// TIA Portal V20 export
FUNCTION_BLOCK "SysCounterFast"   // FB2035, FBD
TITLE = manage a incremental encoder conected to a counter module
{ S7_Optimized_Access := 'TRUE' }
AUTHOR : MiCROTEC
VERSION : 1.6
// -2018.09 : Martin
// -2019.10 : Martin
// stored: AutoNumber false, MemoryReserve 100, SetENOAutomatically false
   VAR_INPUT
      adr { ExternalAccessible := 'False'; ExternalVisible := 'False'; ExternalWritable := 'False'} : HW_IO;   // I/O adresse
      changeDir { ExternalAccessible := 'False'; ExternalVisible := 'False'; ExternalWritable := 'False'} : Bool;   // change direction
      reset { ExternalAccessible := 'False'; ExternalVisible := 'False'; ExternalWritable := 'False'} : Bool;   // reset counter
      calOffset { ExternalAccessible := 'False'; ExternalVisible := 'False'; ExternalWritable := 'False'} : Real;   // offset [mm], the "Reset" will take effect after the offset value
      calGain { ExternalAccessible := 'False'; ExternalVisible := 'False'; ExternalWritable := 'False'} : Real;   // gain
      set { ExternalAccessible := 'False'; ExternalVisible := 'False'; ExternalWritable := 'False'} : Bool;   // set counter on "set value"
      setValue { ExternalAccessible := 'False'; ExternalVisible := 'False'; ExternalWritable := 'False'} : Real;   // set value [mm]
      ack { ExternalAccessible := 'False'; ExternalVisible := 'False'; ExternalWritable := 'False'} : Bool;   // fault acknowledge
      runCheckActive { ExternalAccessible := 'False'; ExternalVisible := 'False'; ExternalWritable := 'False'} : Bool;   // activate plausibility check of encoder value and run signal
      runCheckTime { ExternalAccessible := 'False'; ExternalVisible := 'False'; ExternalWritable := 'False'} : Time := T#3S;   // run signal check fault time
      runCheckDiff { ExternalAccessible := 'False'; ExternalVisible := 'False'; ExternalWritable := 'False'} : Real := 0.5;   // difference value for run check
      runSig { ExternalAccessible := 'False'; ExternalVisible := 'False'; ExternalWritable := 'False'} : Bool;   // run signal for drive
      errOffDelTime { ExternalAccessible := 'False'; ExternalVisible := 'False'; ExternalWritable := 'False'} : Time := T#1S;   // err off delayed time
      limMin { ExternalAccessible := 'False'; ExternalVisible := 'False'; ExternalWritable := 'False'} : Real;   // minimum limit position (0 = deactivated )
      limMax { ExternalAccessible := 'False'; ExternalVisible := 'False'; ExternalWritable := 'False'} : Real;   // maximum limit position (0 = deactivated )
   END_VAR
   VAR_OUTPUT
      comOk { ExternalAccessible := 'False'; ExternalVisible := 'False'; ExternalWritable := 'False'} : Bool;   // communication ok/active
      ready { ExternalAccessible := 'False'; ExternalVisible := 'False'; ExternalWritable := 'False'} : Bool;   // ready to work
      encAct { ExternalAccessible := 'False'; ExternalVisible := 'False'; ExternalWritable := 'False'} : DInt;   // actual position from counter
      delta { ExternalAccessible := 'False'; ExternalVisible := 'False'; ExternalWritable := 'False'} : Real;   // delta in millimeter
      resetPos { ExternalAccessible := 'False'; ExternalVisible := 'False'; ExternalWritable := 'False'} : Real;   // last reset position for the encoder value (ex. division sensor)
      act { ExternalAccessible := 'False'; ExternalVisible := 'False'; ExternalWritable := 'False'} : Real;   // actual position in millimeter
      sync { ExternalAccessible := 'False'; ExternalVisible := 'False'; ExternalWritable := 'False'} : Bool;   // reset puls (division sensor, or generate with offset)
      err { ExternalAccessible := 'False'; ExternalVisible := 'False'; ExternalWritable := 'False'} : Bool;   // fault
      errCom { ExternalAccessible := 'False'; ExternalVisible := 'False'; ExternalWritable := 'False'} : Bool;   // fault communication
      errRdEnc { ExternalAccessible := 'False'; ExternalVisible := 'False'; ExternalWritable := 'False'} : Bool;   // fault encoder from count module
      errRunCheck { ExternalAccessible := 'False'; ExternalVisible := 'False'; ExternalWritable := 'False'} : Bool;   // fault plausibility check run-signal/encoder-value
      errLim { ExternalAccessible := 'False'; ExternalVisible := 'False'; ExternalWritable := 'False'} : Bool;   // fault position is outside from limits
      errOverFlow { ExternalAccessible := 'False'; ExternalVisible := 'False'; ExternalWritable := 'False'} : Bool;   // fault implausible change in encoder value detected (maybe overflow or underflow)
   END_VAR
   VAR_IN_OUT
      Enc : "TypeEncoder";
   END_VAR
   VAR
      var { ExternalAccessible := 'False'; ExternalVisible := 'False'; ExternalWritable := 'False'; S7_SetPoint := 'True'} : "TypeVar";
      T { ExternalAccessible := 'False'; ExternalVisible := 'False'; ExternalWritable := 'False'; S7_SetPoint := 'True'} : Array[1..3] of IEC_TIMER;
      Rd { ExternalAccessible := 'False'; ExternalVisible := 'False'; ExternalWritable := 'False'} : Struct
         cntBit24 : Bool;   // count value
         stsDI1 : Bool;   // DI1 status
         stsDir : Bool;   // direction
         stsDI0 : Bool;   // DI0 status
         err : Bool;   // fault
         stsDI2 : Bool;   // Tm Count: status DI2
         stsReady : Bool;   // ready
         Wd : Bool;   // watchdog if used isochronous mode
         cntValue2 : Byte;   // count value
         cntValue : Word;   // count value
      END_STRUCT;
      encActOld { ExternalAccessible := 'False'; ExternalVisible := 'False'; ExternalWritable := 'False'} : DInt;
      deltaIncOld { ExternalAccessible := 'False'; ExternalVisible := 'False'; ExternalWritable := 'False'} : DInt;
      actualNoOffset { ExternalAccessible := 'False'; ExternalVisible := 'False'; ExternalWritable := 'False'} : Real;
      errLimMin { ExternalAccessible := 'False'; ExternalVisible := 'False'; ExternalWritable := 'False'} : Bool;
      errLimMax { ExternalAccessible := 'False'; ExternalVisible := 'False'; ExternalWritable := 'False'} : Bool;
   END_VAR
   VAR_TEMP
      tempDelta1 : DInt;
      tempRdRetVal : Int;
      tempErrOverFlow : Bool;
   END_VAR
   VAR_TEMP   // added for the SCL form of the ladder/FBD networks
      _w1 : Bool;
      _w2 : Bool;
   END_VAR
BEGIN

REGION Network 1: exit
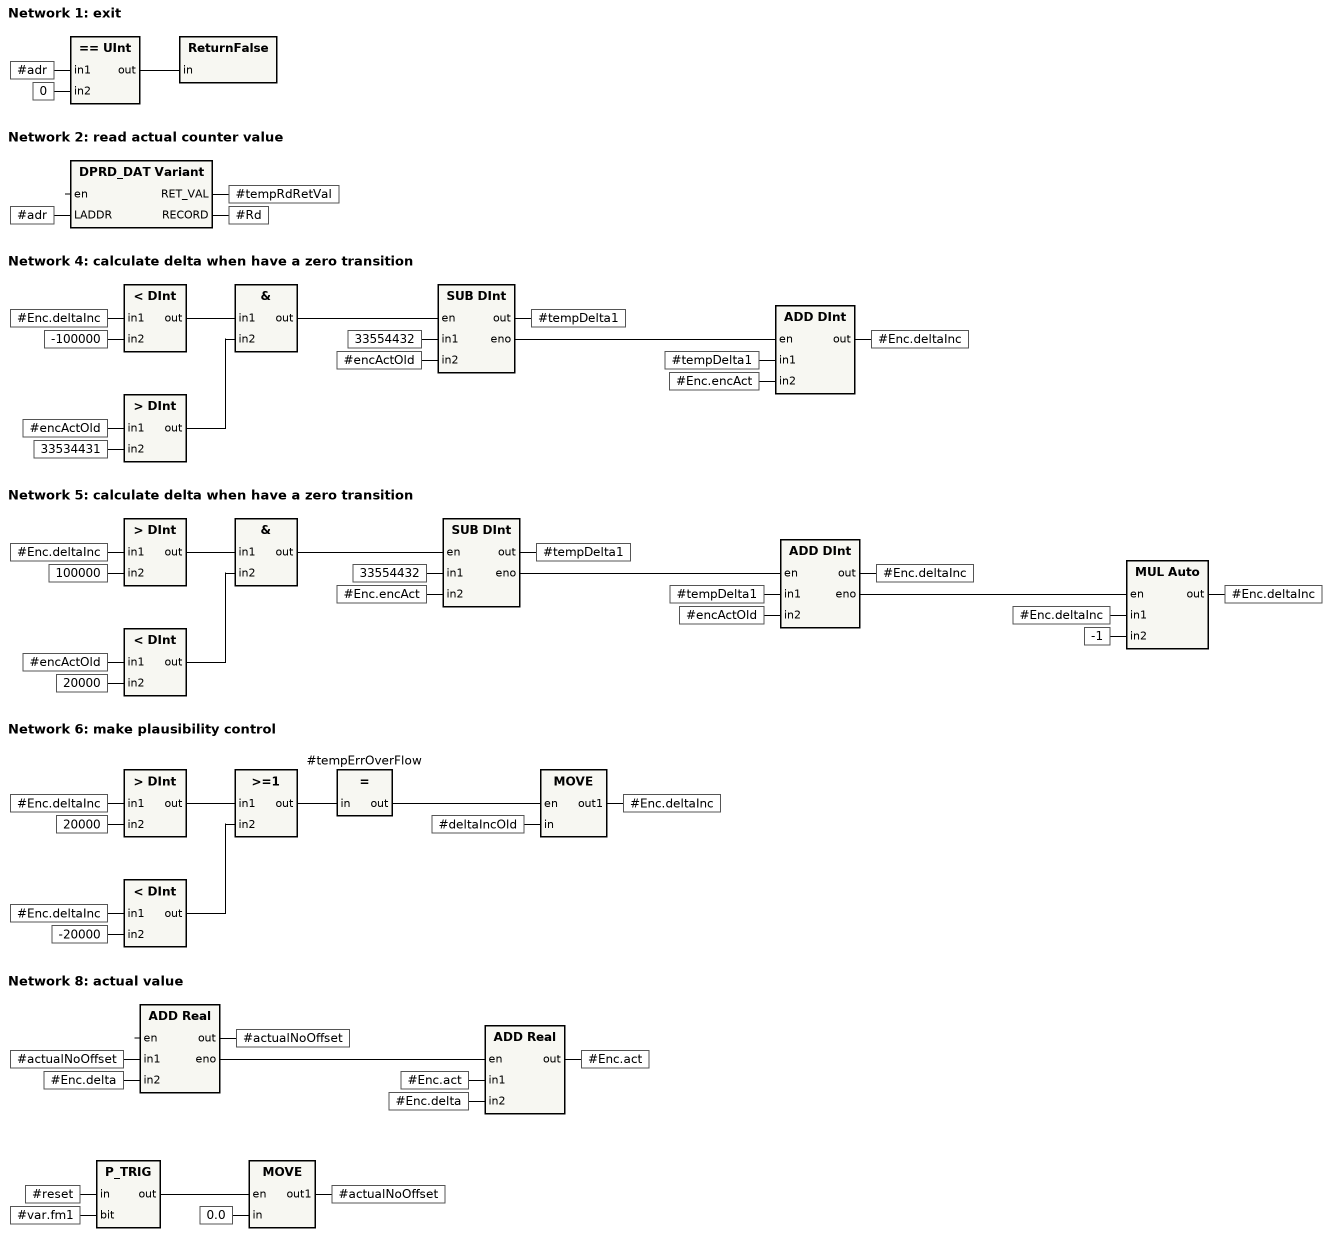
   IF #adr = 0 THEN
       ENO := FALSE;
       RETURN;
   END_IF;
END_REGION

REGION Network 2: read actual counter value
   #tempRdRetVal := DPRD_DAT(LADDR := #adr, RECORD => #Rd);
END_REGION

REGION Network 3 (SCL): read/write values

   #Enc.ready := #Rd.stsReady;
   #Enc.encAct :=  WORD_TO_DWORD(#Rd.cntValue) OR SHL_DWORD(IN:=BYTE_TO_DWORD(#Rd.cntValue2), N:=16);
   #Enc.encAct.%X24 := #Rd.cntBit24;
   #Enc.calOffset := #calOffset;
   #Enc.refPos := #setValue;
   #Enc.limMin := #limMin;
   #Enc.limMax := #limMax;
   #Enc.dirUp := #Rd.stsDir;
   #Enc.dirDn := NOT #Rd.stsDir;

   IF #calGain <> 0.0 THEN
       #Enc.calGain := #calGain;
   ELSE
       #Enc.calGain := 1.0;
   END_IF;

   #Enc.deltaInc := #Enc.encAct - #encActOld;
END_REGION

REGION Network 4: calculate delta when have a zero transition
   // ENO of a box is taken as its EN; it also drops when the box reports an error
   IF (#Enc.deltaInc < (-100000)) AND (#encActOld > 33534431) THEN
       #tempDelta1 := 33554432 - #encActOld;
       #Enc.deltaInc := #tempDelta1 + #Enc.encAct;
   END_IF;
END_REGION

REGION Network 5: calculate delta when have a zero transition
   // ENO of a box is taken as its EN; it also drops when the box reports an error
   IF (#Enc.deltaInc > 100000) AND (#encActOld < 20000) THEN #tempDelta1 := 33554432 - #Enc.encAct; END_IF;
   #_w1 := (#Enc.deltaInc > 100000) AND (#encActOld < 20000);
   IF #_w1 THEN
       #Enc.deltaInc := #tempDelta1 + #encActOld;
       #Enc.deltaInc := #Enc.deltaInc * (-1);
   END_IF;
END_REGION

REGION Network 6: make plausibility control
   #tempErrOverFlow := (#Enc.deltaInc > 20000) OR (#Enc.deltaInc < (-20000));
   IF #tempErrOverFlow THEN #Enc.deltaInc := #deltaIncOld; END_IF;
END_REGION

REGION Network 7 (SCL): increment in mm and actual speed in meter/min
   #Enc.delta := DINT_TO_REAL( #Enc.deltaInc) * #Enc.calGain;
   #Enc.speed := #Enc.speed * 0.9 + (#Enc.delta * 60.0 / "cycle") * 0.1;

   //save old value
   #deltaIncOld := #Enc.deltaInc;
   #encActOld := #Enc.encAct;
END_REGION

REGION Network 8: actual value
   // ENO of a box is taken as its EN; it also drops when the box reports an error
   #actualNoOffset := #actualNoOffset + #Enc.delta;
   #Enc.act := #Enc.act + #Enc.delta;
   #_w1 := #reset AND NOT #var.fm1;   // rising edge
   #var.fm1 := #reset;
   IF #_w1 THEN #actualNoOffset := 0.0; END_IF;
END_REGION

REGION Network 9: virtual reset
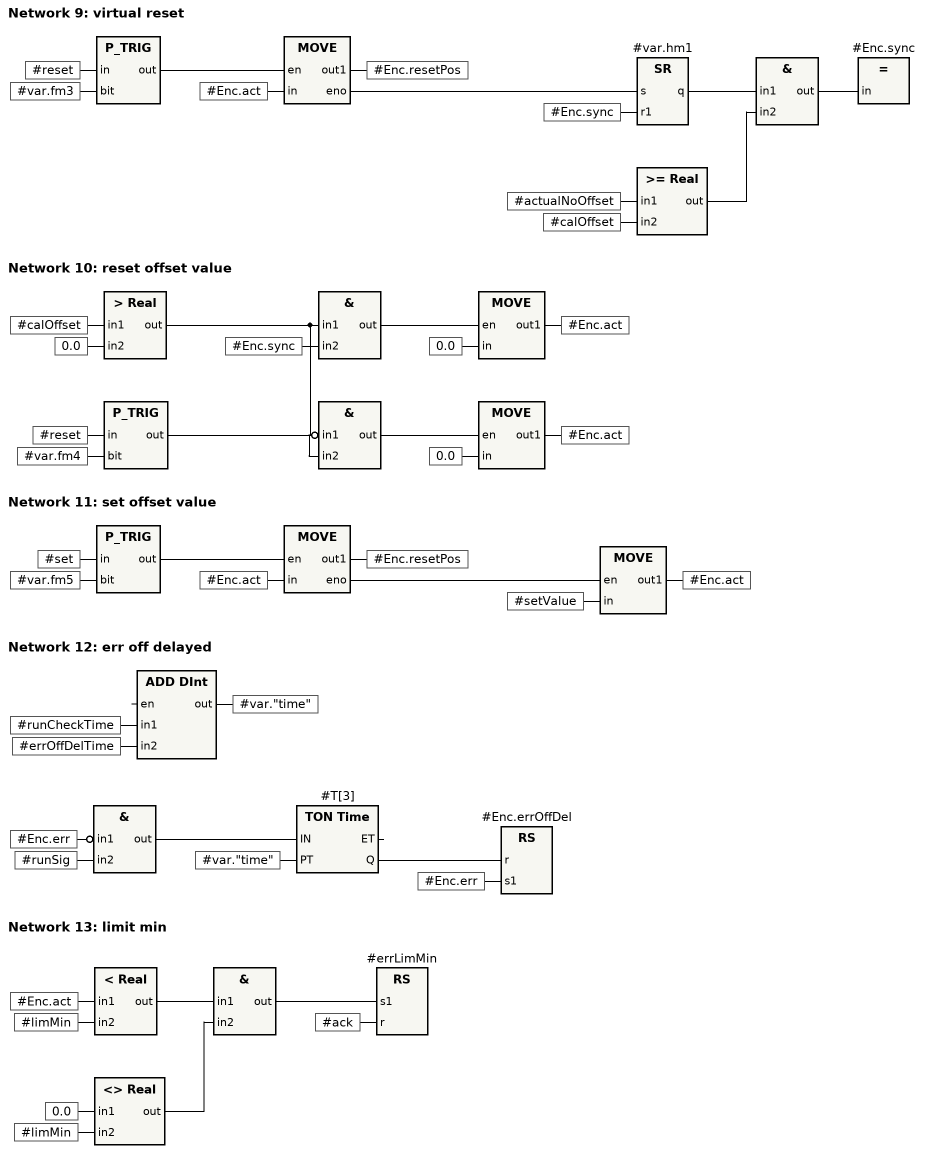
   #_w1 := #reset AND NOT #var.fm3;   // rising edge
   #var.fm3 := #reset;
   IF #_w1 THEN
       #Enc.resetPos := #Enc.act;
       #var.hm1 := TRUE;   // SR flip-flop
   END_IF;
   IF #Enc.sync THEN #var.hm1 := FALSE; END_IF;
   #Enc.sync := #var.hm1 AND (#actualNoOffset >= #calOffset);
END_REGION

REGION Network 10: reset offset value
   #_w1 := #calOffset > 0.0;
   IF #_w1 AND #Enc.sync THEN #Enc.act := 0.0; END_IF;
   #_w2 := #reset AND NOT #var.fm4;   // rising edge
   #var.fm4 := #reset;
   IF NOT #_w1 AND #_w2 THEN #Enc.act := 0.0; END_IF;
END_REGION

REGION Network 11: set offset value
   #_w1 := #set AND NOT #var.fm5;   // rising edge
   #var.fm5 := #set;
   IF #_w1 THEN
       #Enc.resetPos := #Enc.act;
       #Enc.act := #setValue;
   END_IF;
END_REGION

REGION Network 12: err off delayed
   #var."time" := #runCheckTime + #errOffDelTime;
   #T[3].TON(IN := NOT #Enc.err AND #runSig, PT := #var."time");
   IF #T[3].Q THEN
       #Enc.errOffDel := FALSE;   // RS flip-flop
   END_IF;
   IF #Enc.err THEN #Enc.errOffDel := TRUE; END_IF;
END_REGION

REGION Network 13: limit min
   IF #ack THEN
       #errLimMin := FALSE;   // RS flip-flop
   END_IF;
   IF (#Enc.act < #limMin) AND (0.0 <> #limMin) THEN #errLimMin := TRUE; END_IF;
END_REGION

REGION Network 14: limit max
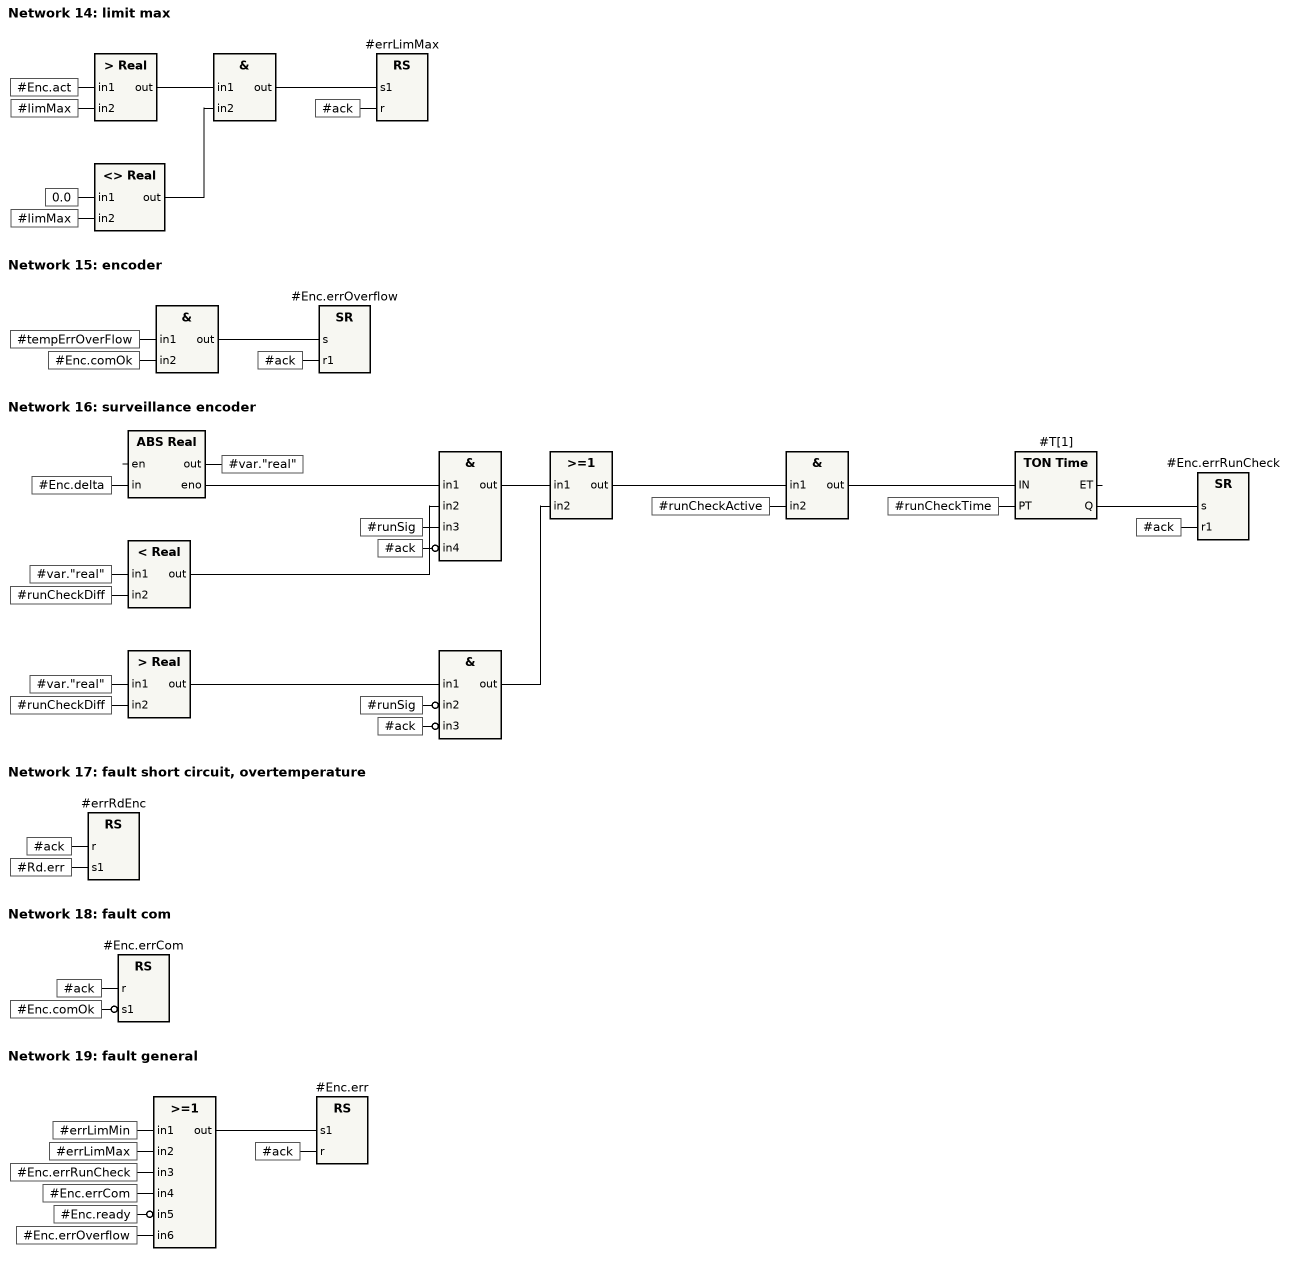
   IF #ack THEN
       #errLimMax := FALSE;   // RS flip-flop
   END_IF;
   IF (#Enc.act > #limMax) AND (0.0 <> #limMax) THEN #errLimMax := TRUE; END_IF;
END_REGION

REGION Network 15: encoder
   IF #tempErrOverFlow AND #Enc.comOk THEN
       #Enc.errOverflow := TRUE;   // SR flip-flop
   END_IF;
   IF #ack THEN #Enc.errOverflow := FALSE; END_IF;
END_REGION

REGION Network 16: surveillance encoder
   #var."real" := ABS(#Enc.delta);
   #T[1].TON(IN := (((#var."real" < #runCheckDiff) AND #runSig AND NOT #ack) OR ((#var."real" > #runCheckDiff) AND NOT #runSig AND NOT #ack)) AND #runCheckActive,
             PT := #runCheckTime);
   IF #T[1].Q THEN
       #Enc.errRunCheck := TRUE;   // SR flip-flop
   END_IF;
   IF #ack THEN #Enc.errRunCheck := FALSE; END_IF;
END_REGION

REGION Network 17: fault short circuit, overtemperature
   IF #ack THEN
       #errRdEnc := FALSE;   // RS flip-flop
   END_IF;
   IF #Rd.err THEN #errRdEnc := TRUE; END_IF;
END_REGION

REGION Network 18: fault com
   IF #ack THEN
       #Enc.errCom := FALSE;   // RS flip-flop
   END_IF;
   IF NOT #Enc.comOk THEN #Enc.errCom := TRUE; END_IF;
END_REGION

REGION Network 19: fault general
   IF #ack THEN
       #Enc.err := FALSE;   // RS flip-flop
   END_IF;
   IF #errLimMin OR #errLimMax OR #Enc.errRunCheck OR #Enc.errCom OR NOT #Enc.ready OR #Enc.errOverflow THEN
       #Enc.err := TRUE;
   END_IF;
END_REGION

REGION Network 20: error number counter [1-50]
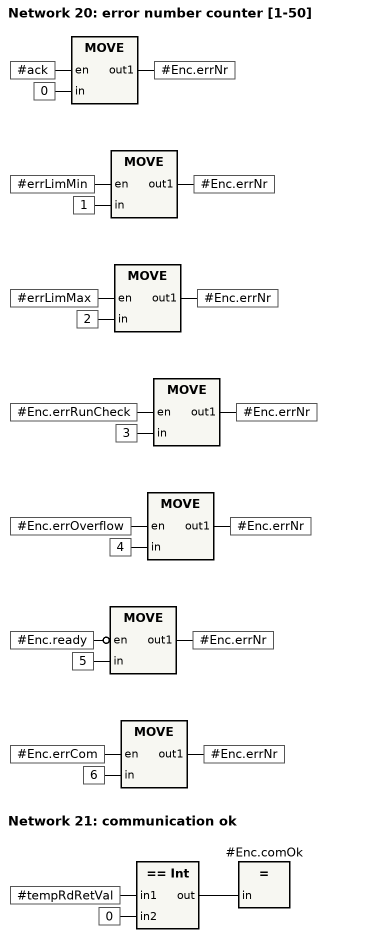
   IF #ack THEN #Enc.errNr := 0; END_IF;
   IF #errLimMin THEN #Enc.errNr := 1; END_IF;
   IF #errLimMax THEN #Enc.errNr := 2; END_IF;
   IF #Enc.errRunCheck THEN #Enc.errNr := 3; END_IF;
   IF #Enc.errOverflow THEN #Enc.errNr := 4; END_IF;
   IF NOT #Enc.ready THEN #Enc.errNr := 5; END_IF;
   IF #Enc.errCom THEN #Enc.errNr := 6; END_IF;
END_REGION

REGION Network 21: communication ok
   #Enc.comOk := #tempRdRetVal = 0;
END_REGION

REGION Network 22 (SCL): write to outputs and encoder data
   #comOk := #Enc.comOk;
   #ready := #Enc.ready;

   #encAct := #Enc.encAct;
   #delta := #Enc.delta;
   #act := #Enc.act ;
   #resetPos := #Enc.resetPos;
   #sync := #Enc.sync;

   #err := #Enc.err;
   #errCom := #Enc.errCom ;
   #errRunCheck := #Enc.errRunCheck ;
   #errLim := #errLimMin OR #errLimMax;
   #errOverFlow := #Enc.errOverflow;

   #Enc.errLim := #errLimMin OR #errLimMax;
   //#Enc.refOk := NOT #Enc.errLim;
END_REGION
END_FUNCTION_BLOCK
